FUNCTION_BLOCK FMA_TRIGGER (* Composite Function Block Type *)
  (* Standard: 61499-2 *)
  (* Version 1.0, 2019-04-11, adeel *)
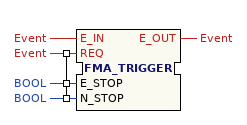
  EVENT_INPUT
    E_IN;
    REQ WITH E_STOP, N_STOP; (* Normal Execution Request *)
  END_EVENT
  EVENT_OUTPUT
    E_OUT;
  END_EVENT
  VAR_INPUT
    E_STOP : BOOL;
    N_STOP : BOOL;
  END_VAR
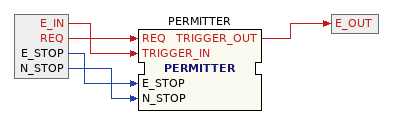
  FBS
    PERMITTER : PERMITTER;
  END_FBS
  EVENT_CONNECTIONS
    REQ TO PERMITTER.REQ;
    E_IN TO PERMITTER.TRIGGER_IN;
    PERMITTER.TRIGGER_OUT TO E_OUT;
  END_CONNECTIONS
  DATA_CONNECTIONS
    E_STOP TO PERMITTER.E_STOP;
    N_STOP TO PERMITTER.N_STOP;
  END_CONNECTIONS
END_FUNCTION_BLOCK
